{attribute 'qualified_only'}
{attribute 'strict'}
TYPE E_ControlBoxMode :
(
	Off,
	Auto,
	Manual
);
END_TYPE

(* stored: Version 1.1.0.1, ProductVersion 3.1.4024.12
   DUT E_ControlBoxMode: Id {85245e45-3f8f-4c02-a25d-60372deec6c5} *)
